(* PLC project drill, Dassault Systèmes ControlBuild 2024x Refresh1 *)
(* stored: creationDateTime 2024-03-06T09:36:38-01:00 *)

CONFIGURATION drill
  VAR_GLOBAL
    generalPanel/batchCycle : BOOL := true;
    generalPanel/cycleSwitch/leftVariable : BOOL := false;
    generalPanel/emergencyStop/PBLogic : BOOL := false;
    functional/descent/motorOfTurret/motor/nominalTime : REAL := 0.05;
    functional/descent/motorOfTurret/motor/nominalLowSpeed : REAL := 100.0;
    functional/descent/motorOfTurret/motor/nominalHighSpeed : REAL := 200.0;
    functional/clamping/leftJack/jack/time2extend : REAL := 1.0;
    functional/clamping/rightJack/jack/time2extend : REAL := 1.0;
  END_VAR
END_CONFIGURATION
